Fanuc KAREL source: ka00121.KL

PROGRAM KA00121
%NOLOCKGROUP
VAR
SRC : ARRAY[2] OF BYTE
DST:INTEGER
BEGIN
SRC[1]=2
DST=SRC[1]
END KA00121
